# B&R Automation Studio project BR_Lab2
Automation Studio 4.5.2.102

## Logical view

### Library Logical/Library (ANSIC)

#### Library.fun
```iecst
{REDUND_ERROR} {REDUND_UNREPLICABLE} FUNCTION_BLOCK DriveStateMachine (*TODO: Add your comment here*) (*$GROUP=User,$CAT=User,$GROUPICON=User.png,$CATICON=User.png*)
	VAR_INPUT
		state : {REDUND_UNREPLICABLE} UINT;
		enable : {REDUND_UNREPLICABLE} BOOL;
	END_VAR
	VAR_OUTPUT
		command : {REDUND_UNREPLICABLE} UINT;
		speed : {REDUND_UNREPLICABLE} INT;
	END_VAR
	VAR
		mask : {REDUND_UNREPLICABLE} UINT;
	END_VAR
END_FUNCTION_BLOCK

{REDUND_ERROR} {REDUND_UNREPLICABLE} FUNCTION_BLOCK DoorStateMachine (*TODO: Add your comment here*) (*$GROUP=User,$CAT=User,$GROUPICON=User.png,$CATICON=User.png*)
	VAR_INPUT
		state : {REDUND_UNREPLICABLE} UINT;
		sw1 : {REDUND_UNREPLICABLE} BOOL;
		sw2 : {REDUND_UNREPLICABLE} BOOL;
		sw3 : {REDUND_UNREPLICABLE} BOOL;
		sw4 : {REDUND_UNREPLICABLE} BOOL;
		direction : {REDUND_UNREPLICABLE} BOOL;
	END_VAR
	VAR_OUTPUT
		speed : {REDUND_UNREPLICABLE} INT;
	END_VAR
END_FUNCTION_BLOCK

{REDUND_ERROR} {REDUND_UNREPLICABLE} FUNCTION_BLOCK LedStateMachine (*TODO: Add your comment here*) (*$GROUP=User,$CAT=User,$GROUPICON=User.png,$CATICON=User.png*)
	VAR_INPUT
		state : {REDUND_UNREPLICABLE} UINT;
	END_VAR
	VAR_OUTPUT
		led1 : {REDUND_UNREPLICABLE} BOOL;
		led2 : {REDUND_UNREPLICABLE} BOOL;
		led3 : {REDUND_UNREPLICABLE} BOOL;
		led4 : {REDUND_UNREPLICABLE} BOOL;
		timer : {REDUND_UNREPLICABLE} INT;
	END_VAR
END_FUNCTION_BLOCK
```

#### DoorStateMachine.c
```c
#include <bur/plctypes.h>
#ifdef __cplusplus
	extern "C"
	{
#endif
	#include "Library.h"
#ifdef __cplusplus
	};
#endif
/* TODO: Add your comment here */
void DoorStateMachine(struct DoorStateMachine* inst)
{
	/*TODO: Add your code here*/
	switch(inst->state)
	{
		case ST_INIT:
			{
				inst->state = ST_UNKNOWN;
				break;
			}

		case ST_UNKNOWN:
			{
				if(inst->direction == 0) {
					inst->state = ST_OPEN;
				}
				if (inst->direction == 1) {
					inst->state = ST_CLOSE;
				}
				break;
			}

		case ST_OPEN:
			{
				inst->speed = 0;
				if(inst->direction == 0) {
					inst->state=ST_ACC_POS;
				}
				break;
			}

		case ST_ACC_POS:
			{
				inst->speed = 150;
				if(inst->sw2) {
					inst->state = ST_POS;
				}
				if (inst->direction == 1) {
					inst->state = ST_DEC_NEG;
				}
				break;
			}

		case ST_POS:
			{
				inst->speed = 900;
				if(inst->sw3) {
					inst->state = ST_DEC_POS;
				}
				if(inst->direction == 1) {
					inst->state = ST_NEG;
				}
			}
			break;

		case ST_DEC_POS:
			{
				inst->speed = 150;
				if(inst->sw4) {
					inst->state = ST_CLOSE;
				}
				break;
			}

		case ST_CLOSE:
			{
				inst->speed = 0;
				if(inst->direction == 1) {
					inst->state=ST_ACC_NEG;
				}
				break;
			}

		case ST_ACC_NEG:
			{
				inst->speed = -150;
				if(inst->sw3) {
					inst->state = ST_NEG;
				}
				if (inst->direction == 0) {
					inst->state = ST_DEC_POS;
				}
				break;
			}

		case ST_NEG:
			{
				inst->speed = -900;
				if(inst->sw2) {
					inst->state = ST_DEC_NEG;
				}
				if(inst->direction == 0) {
					inst->state = ST_POS;
				}
				break;
			}

		case ST_DEC_NEG:
			{
				inst->speed = -150;
				if(inst->sw1) {
					inst->state = ST_OPEN;
				}
				break;
			}
	}
}
```

#### DriveStateMachine.c
```c
#include <bur/plctypes.h>
#ifdef __cplusplus
	extern "C"
	{
#endif
	#include "Library.h"
#ifdef __cplusplus
	};
#endif

void DriveStateMachine(struct DriveStateMachine* inst)
{
    UINT mask = inst->state & 0x6f;
	if(!inst->enable)
	{
		inst->command = CMD_SHUTDOWN;
	}
	else
	{
		switch (mask)
		{
			case STATE_DISABLED:
				inst->command = CMD_SHUTDOWN;
				break;

			case STATE_READY:
				inst->command = CMD_ENABLE;
				break;

			case STATE_SWITCHED_ON:
				inst->command = CMD_SWITCH_ON;
				break;
		}
	}
}
```

### Program Logical/Program (ANSIC)

#### Variables.var
```iecst
VAR
	doorSM : {REDUND_UNREPLICABLE} DoorStateMachine := (0);
	ledSM : {REDUND_UNREPLICABLE} LedStateMachine := (0);
	driveSM : {REDUND_UNREPLICABLE} DriveStateMachine := (0);
END_VAR
```

#### Main.c
```c
#include <bur/plctypes.h>

#ifdef _DEFAULT_INCLUDES
	#include <AsDefault.h>
#endif

void _INIT ProgramInit(void)
{
    driveSM.enable=1;
}

void _CYCLIC ProgramCyclic(void)
{
    DoorStateMachine(&doorSM);
    driveSM.speed = doorSM.speed;
    DriveStateMachine(&driveSM);
    ledSM.state = doorSM.state;
    LedStateMachine(&ledSM);
}

void _EXIT ProgramExit(void)
{

}
```

Listed in the project but not available here: Logical/Global.typ, Logical/Global.var, Logical/Libraries, Logical/ncsdcctrl, Logical/acp10etxen, Logical/gAxis01obj
